# B&R Automation Studio project DO_Workshop
Automation Studio 4.9

## Configuration Config1

CPU X20CP1684, AutomationRuntime E4.93, Build 4.1.2, Vc V4.72.6

### Task classes (Cpu.sw)
```
Cyclic#4:
  Merge <- Merge.prg
Libraries: AsBrStr
```

### Hardware
```
X20CP1684 : X20CP1684 v1.7.2.0
```

## Logical view

Binary libraries used (declarations not repeated): operator, runtime, astime, AsIecCon, AsBrStr


### Program Logical/Merge (IEC)

#### Merge.st - Init, cyclic, exit code
```iecst
PROGRAM _INIT

END_PROGRAM

PROGRAM _CYCLIC

//	Output1		:= Input1;

	// TODO - Enter your line of code on the line below.  Perform math operations on Input1 and assign to Output1
	Output1 := Input1 * 2;

END_PROGRAM

PROGRAM _EXIT
	(* Insert code here *)

END_PROGRAM
```

#### Variables.var - Local variables
```iecst
VAR
	Output1 : REAL;
	Input1 : REAL;
END_VAR
```

#### Merge_BACKUP_2007.st - not listed in the package file held
```iecst
PROGRAM _INIT

END_PROGRAM

PROGRAM _CYCLIC

	Output1		:= Input1;

	// TODO - Enter your line of code on the line below.  Perform math operations on Input1 and assign to Output1
<<<<<<< HEAD
	Output1		:= Input1 * 100.0 / 65.0;

=======
	Output1     := Input1*500/3;
>>>>>>> origin/Feature/jess
END_PROGRAM

PROGRAM _EXIT
	(* Insert code here *)

END_PROGRAM
```

#### Merge_BASE_2007.st - not listed in the package file held
```iecst
PROGRAM _INIT

END_PROGRAM

PROGRAM _CYCLIC

	Output1		:= Input1;

	// TODO - Enter your line of code on the line below.  Perform math operations on Input1 and assign to Output1

END_PROGRAM

PROGRAM _EXIT
	(* Insert code here *)

END_PROGRAM
```

#### Merge_LOCAL_2007.st - not listed in the package file held
```iecst
PROGRAM _INIT

END_PROGRAM

PROGRAM _CYCLIC

	Output1		:= Input1;

	// TODO - Enter your line of code on the line below.  Perform math operations on Input1 and assign to Output1
	Output1		:= Input1 * 100.0 / 65.0;

END_PROGRAM

PROGRAM _EXIT
	(* Insert code here *)

END_PROGRAM
```

#### Merge_REMOTE_2007.st - not listed in the package file held
```iecst
PROGRAM _INIT

END_PROGRAM

PROGRAM _CYCLIC

	Output1		:= Input1;

	// TODO - Enter your line of code on the line below.  Perform math operations on Input1 and assign to Output1
	Output1     := Input1*500/3;
END_PROGRAM

PROGRAM _EXIT
	(* Insert code here *)

END_PROGRAM
```

Listed in the project but not available here: Logical/Global.typ, Logical/Global.var, Logical/Merge/Types.typ
